// TIA Portal V17 export
// export: Created 2024-01-30T08:49:17.494963Z, ExportSetting WithDefaults, DisplayName Totally Integrated Automation Portal, DisplayVersion V17 Update 6, DisplayName TIA Portal Openness, DisplayVersion V17 Update 6, DisplayName TIA Portal Version Control Interface, DisplayVersion V17, DisplayName STEP 7 Professional, DisplayVersion V17 Update 6, DisplayName STEP 7 Safety, DisplayVersion V17 Update 6, DisplayName WinCC Advanced, DisplayVersion V17 Update 6
TYPE "UDT_RS232_SEND_DATA"
// stored: IsFailsafeCompliant false
   STRUCT
      Data : Array[0..23] of Byte;
   END_STRUCT;
END_TYPE
